// Mitsubishi GX Works2 project: FINAL   PLC: Q03UDV

PROGRAM MAIN
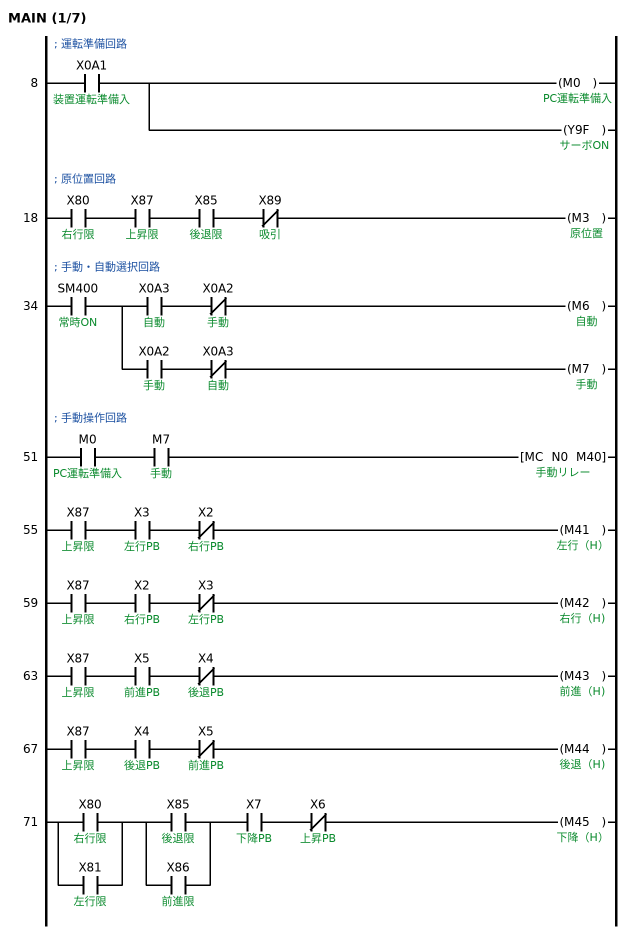
; 運転準備回路
8     LD      X0A1  ; 装置運転準備入
      OUT     M0  ; PC運転準備入
      OUT     Y9F  ; サーボON
; 原位置回路
18    LD      X80  ; 右行限
      AND     X87  ; 上昇限
      AND     X85  ; 後退限
      ANI     X89  ; 吸引
      OUT     M3  ; 原位置
; 手動・自動選択回路
34    LD      SM400  ; 常時ON
      MPS
      AND     X0A3  ; 自動
      ANI     X0A2  ; 手動
      OUT     M6  ; 自動
      MPP
      AND     X0A2  ; 手動
      ANI     X0A3  ; 自動
      OUT     M7  ; 手動
; 手動操作回路
51    LD      M0  ; PC運転準備入
      AND     M7  ; 手動
      MC      N0 M40  ; 手動リレー
55    LD      X87  ; 上昇限
      AND     X3  ; 左行PB
      ANI     X2  ; 右行PB
      OUT     M41  ; 左行（H）
59    LD      X87  ; 上昇限
      AND     X2  ; 右行PB
      ANI     X3  ; 左行PB
      OUT     M42  ; 右行（H)
63    LD      X87  ; 上昇限
      AND     X5  ; 前進PB
      ANI     X4  ; 後退PB
      OUT     M43  ; 前進（H)
67    LD      X87  ; 上昇限
      AND     X4  ; 後退PB
      ANI     X5  ; 前進PB
      OUT     M44  ; 後退（H)
71    LD      X80  ; 右行限
      OR      X81  ; 左行限
      LD      X85  ; 後退限
      OR      X86  ; 前進限
      ANB
      AND     X7  ; 下降PB
      ANI     X6  ; 上昇PB
      OUT     M45  ; 下降（H）
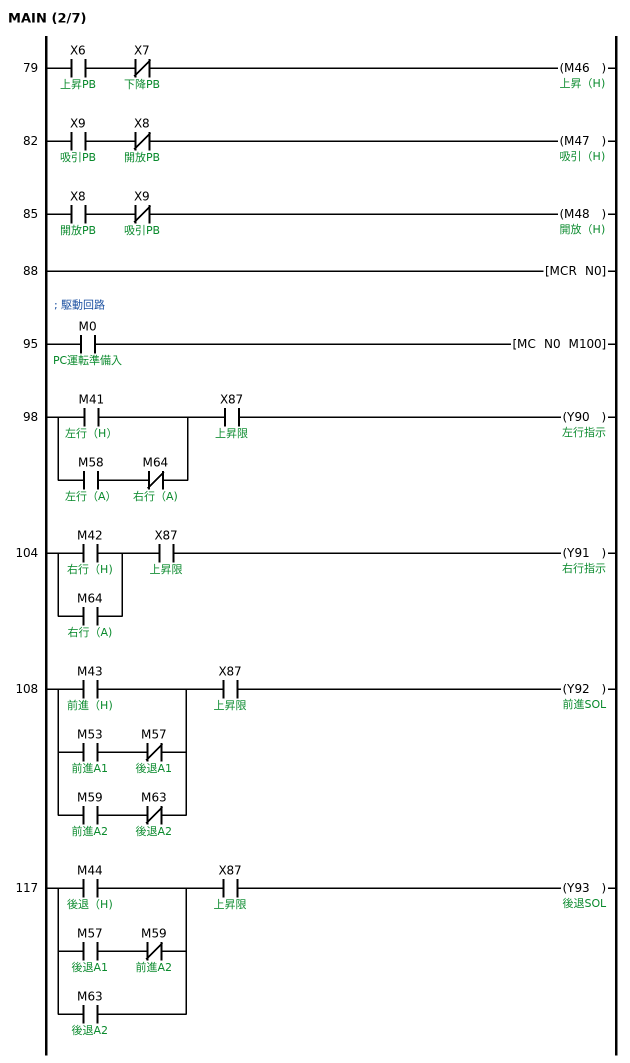
79    LD      X6  ; 上昇PB
      ANI     X7  ; 下降PB
      OUT     M46  ; 上昇（H)
82    LD      X9  ; 吸引PB
      ANI     X8  ; 開放PB
      OUT     M47  ; 吸引（H)
85    LD      X8  ; 開放PB
      ANI     X9  ; 吸引PB
      OUT     M48  ; 開放（H)
88    MCR     N0
; 駆動回路
95    LD      M0  ; PC運転準備入
      MC      N0 M100
98    LD      M41  ; 左行（H）
      LD      M58  ; 左行（A）
      ANI     M64  ; 右行（A)
      ORB
      AND     X87  ; 上昇限
      OUT     Y90  ; 左行指示
104   LD      M42  ; 右行（H)
      OR      M64  ; 右行（A)
      AND     X87  ; 上昇限
      OUT     Y91  ; 右行指示
108   LD      M43  ; 前進（H)
      LD      M53  ; 前進A1
      ANI     M57  ; 後退A1
      ORB
      LD      M59  ; 前進A2
      ANI     M63  ; 後退A2
      ORB
      AND     X87  ; 上昇限
      OUT     Y92  ; 前進SOL
117   LD      M44  ; 後退（H)
      LD      M57  ; 後退A1
      ANI     M59  ; 前進A2
      ORB
      OR      M63  ; 後退A2
      AND     X87  ; 上昇限
      OUT     Y93  ; 後退SOL
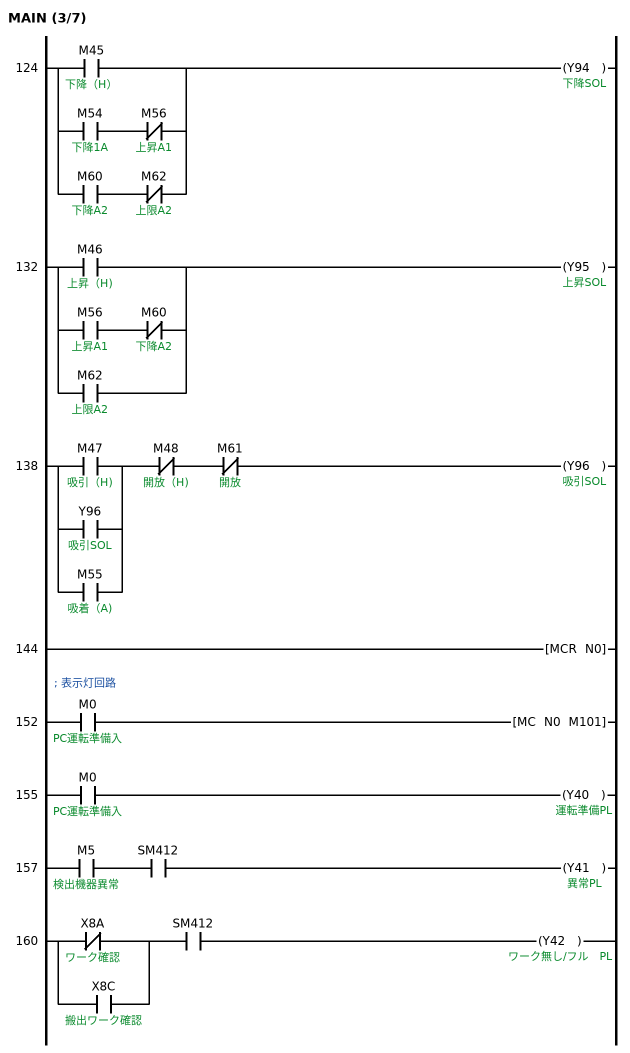
124   LD      M45  ; 下降（H）
      LD      M54  ; 下降1A
      ANI     M56  ; 上昇A1
      ORB
      LD      M60  ; 下降A2
      ANI     M62  ; 上限A2
      ORB
      OUT     Y94  ; 下降SOL
132   LD      M46  ; 上昇（H)
      LD      M56  ; 上昇A1
      ANI     M60  ; 下降A2
      ORB
      OR      M62  ; 上限A2
      OUT     Y95  ; 上昇SOL
138   LD      M47  ; 吸引（H)
      OR      Y96  ; 吸引SOL
      OR      M55  ; 吸着（A)
      ANI     M48  ; 開放（H)
      ANI     M61  ; 開放
      OUT     Y96  ; 吸引SOL
144   MCR     N0
; 表示灯回路
152   LD      M0  ; PC運転準備入
      MC      N0 M101
155   LD      M0  ; PC運転準備入
      OUT     Y40  ; 運転準備PL
157   LD      M5  ; 検出機器異常
      AND     SM412
      OUT     Y41  ; 異常PL
160   LDI     X8A  ; ワーク確認
      OR      X8C  ; 搬出ワーク確認
      AND     SM412
      OUT     Y42  ; ワーク無し/フル　PL
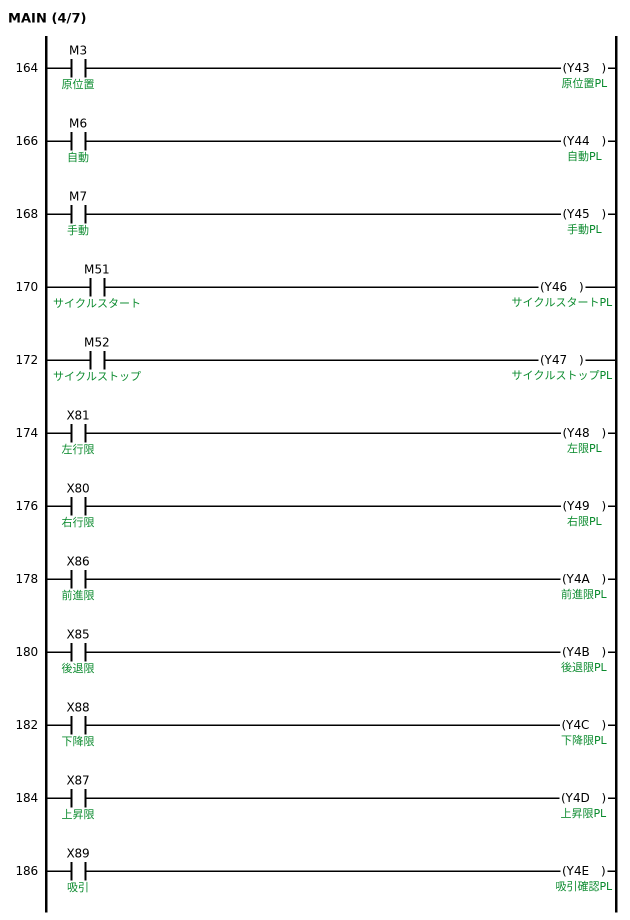
164   LD      M3  ; 原位置
      OUT     Y43  ; 原位置PL
166   LD      M6  ; 自動
      OUT     Y44  ; 自動PL
168   LD      M7  ; 手動
      OUT     Y45  ; 手動PL
170   LD      M51  ; サイクルスタート
      OUT     Y46  ; サイクルスタートPL
172   LD      M52  ; サイクルストップ
      OUT     Y47  ; サイクルストップPL
174   LD      X81  ; 左行限
      OUT     Y48  ; 左限PL
176   LD      X80  ; 右行限
      OUT     Y49  ; 右限PL
178   LD      X86  ; 前進限
      OUT     Y4A  ; 前進限PL
180   LD      X85  ; 後退限
      OUT     Y4B  ; 後退限PL
182   LD      X88  ; 下降限
      OUT     Y4C  ; 下降限PL
184   LD      X87  ; 上昇限
      OUT     Y4D  ; 上昇限PL
186   LD      X89  ; 吸引
      OUT     Y4E  ; 吸引確認PL
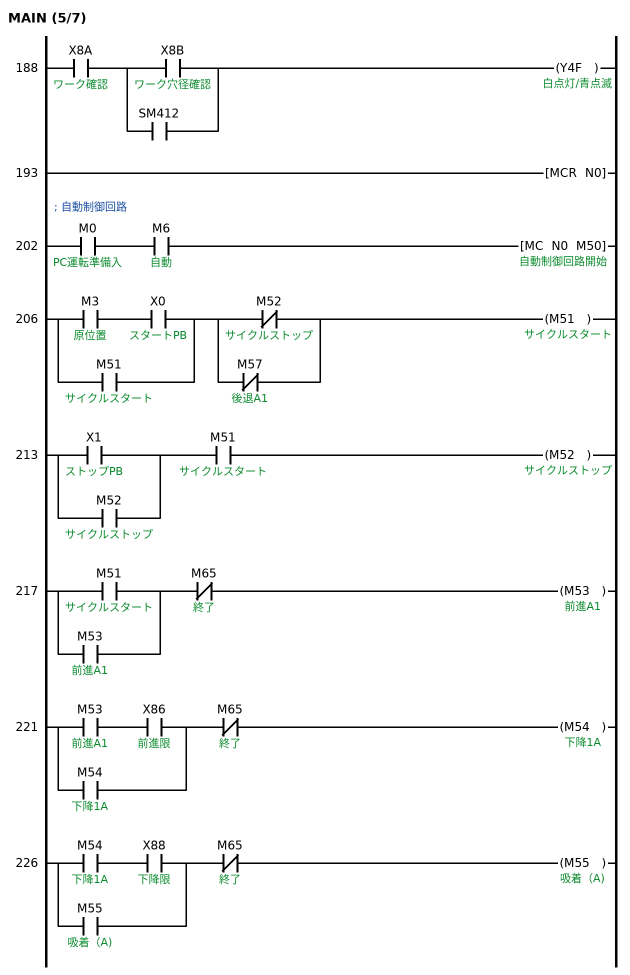
188   LD      X8A  ; ワーク確認
      LD      X8B  ; ワーク穴径確認
      OR      SM412
      ANB
      OUT     Y4F  ; 白点灯/青点滅
193   MCR     N0
; 自動制御回路
202   LD      M0  ; PC運転準備入
      AND     M6  ; 自動
      MC      N0 M50  ; 自動制御回路開始
206   LD      M3  ; 原位置
      AND     X0  ; スタートPB
      OR      M51  ; サイクルスタート
      LDI     M52  ; サイクルストップ
      ORI     M57  ; 後退A1
      ANB
      OUT     M51  ; サイクルスタート
213   LD      X1  ; ストップPB
      OR      M52  ; サイクルストップ
      AND     M51  ; サイクルスタート
      OUT     M52  ; サイクルストップ
217   LD      M51  ; サイクルスタート
      OR      M53  ; 前進A1
      ANI     M65  ; 終了
      OUT     M53  ; 前進A1
221   LD      M53  ; 前進A1
      AND     X86  ; 前進限
      OR      M54  ; 下降1A
      ANI     M65  ; 終了
      OUT     M54  ; 下降1A
226   LD      M54  ; 下降1A
      AND     X88  ; 下降限
      OR      M55  ; 吸着（A)
      ANI     M65  ; 終了
      OUT     M55  ; 吸着（A)
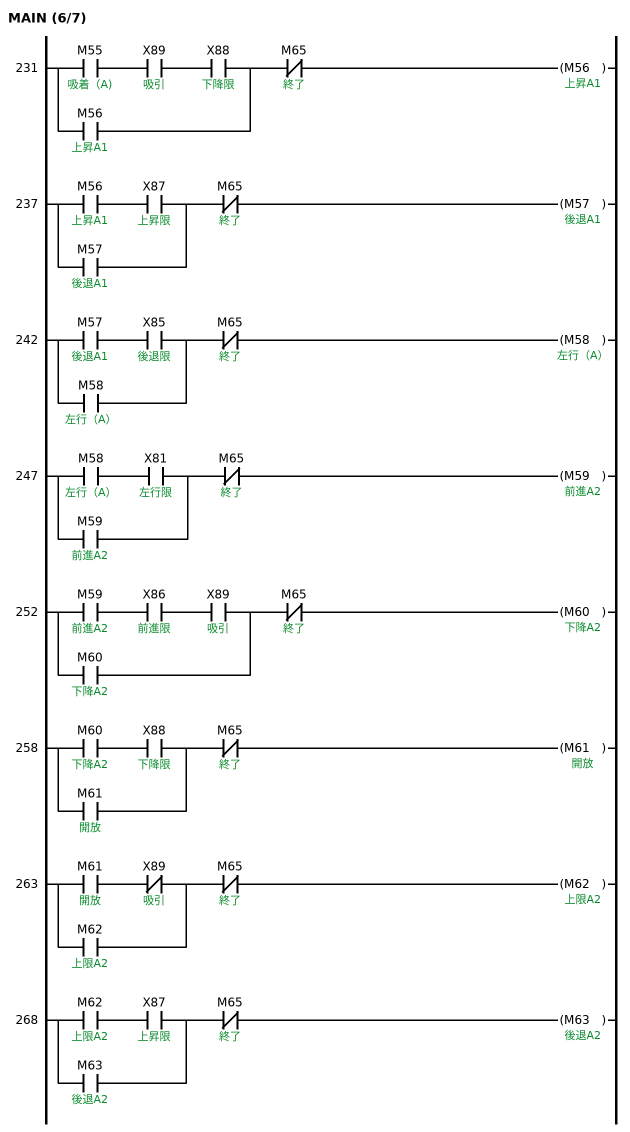
231   LD      M55  ; 吸着（A)
      AND     X89  ; 吸引
      AND     X88  ; 下降限
      OR      M56  ; 上昇A1
      ANI     M65  ; 終了
      OUT     M56  ; 上昇A1
237   LD      M56  ; 上昇A1
      AND     X87  ; 上昇限
      OR      M57  ; 後退A1
      ANI     M65  ; 終了
      OUT     M57  ; 後退A1
242   LD      M57  ; 後退A1
      AND     X85  ; 後退限
      OR      M58  ; 左行（A）
      ANI     M65  ; 終了
      OUT     M58  ; 左行（A）
247   LD      M58  ; 左行（A）
      AND     X81  ; 左行限
      OR      M59  ; 前進A2
      ANI     M65  ; 終了
      OUT     M59  ; 前進A2
252   LD      M59  ; 前進A2
      AND     X86  ; 前進限
      AND     X89  ; 吸引
      OR      M60  ; 下降A2
      ANI     M65  ; 終了
      OUT     M60  ; 下降A2
258   LD      M60  ; 下降A2
      AND     X88  ; 下降限
      OR      M61  ; 開放
      ANI     M65  ; 終了
      OUT     M61  ; 開放
263   LD      M61  ; 開放
      ANI     X89  ; 吸引
      OR      M62  ; 上限A2
      ANI     M65  ; 終了
      OUT     M62  ; 上限A2
268   LD      M62  ; 上限A2
      AND     X87  ; 上昇限
      OR      M63  ; 後退A2
      ANI     M65  ; 終了
      OUT     M63  ; 後退A2
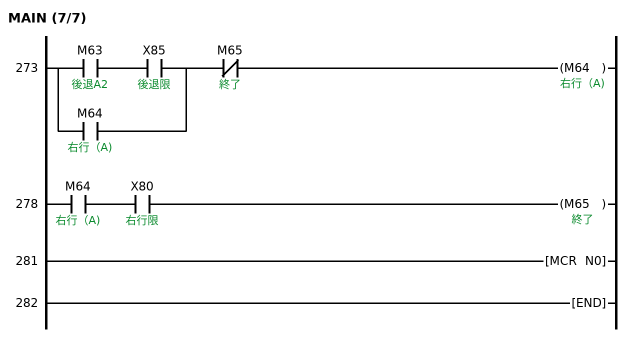
273   LD      M63  ; 後退A2
      AND     X85  ; 後退限
      OR      M64  ; 右行（A)
      ANI     M65  ; 終了
      OUT     M64  ; 右行（A)
278   LD      M64  ; 右行（A)
      AND     X80  ; 右行限
      OUT     M65  ; 終了
281   MCR     N0
282   END
END_PROGRAM

// device comments not shown above
X0F  ; リセッ
